(* CODESYS project projeto_final.project

Project tree, tasks and I/O mapping:
  Device : CODESYS Control Win V3, 3S - Smart Software Solutions GmbH, version 3.5.3.50
    application Application
      libraries: Standard, 3.5.2.0 (System)
      task MainTask (cyclic, interval t#20ms, priority 1) calls liga_desliga, projeto_final
      task simula_vagao (cyclic, interval t#10ms, priority 1) calls simula_vagao_descarrega
      task simula_ventilacao (freewheeling, priority 1) calls simula_SA_01_02_ventilacao
      task simula_SA_carregamento (cyclic, interval t#10ms, priority 1) calls simula_SA_01_carregando
      task simula_descarregamento (cyclic, interval t#20ms, priority 1) calls simula_descarga
      program projeto_final [FBD]
      program liga_desliga [LD]
      function block TR_01_transportador_entrada [SFC]: Receber_graos_active, Transfere_graos_active, Passo_inicial_active, Ativa_transferencia_active
      function block vagao_graneleiro [SFC]: Step0_active, Chave_ligada_active, Step1_active, Step2_active, Inicio_active
      function block MG_01_desviador_mangueira [LD]
      function block SA_01_silo_armazenamento [SFC]: Passo_inicial_active, Carrega_silo_active, Descarrega_silo_active, Passo_auxiliar_active, Transfere_moega_active, Liga_alimentador_active
      function block SA_01_02_nivel_silo [FBD]
      program simula_vagao_descarrega [ST]
      program simula_SA_01_02_ventilacao [LD]
      program simula_SA_01_carregando [ST]
      function block SA_02_silo_armazenamento [SFC]: Passo_inicial_active, Passo_auxiliar_active, Carrega_silo_active, Descarrega_silo_active
      program simula_descarga [ST]
  global variables GVL
*)

// GVL
VAR_GLOBAL
	// liga e desliga
	liga        : BOOL;
	liga_local  : BOOL;
	liga_remoto : BOOL;
	seletor_modo: BOOL; // 1 = local e 0 = remoto
	
	// vagao granaleiro
	vagao_chave              : BOOL; // indica que o vagao esta posicionado
	vagao_descarrega         : BOOL; // recebe comando do sistema de supervisao para descarregar
	vagao_capacidade         : INT;  // kg
	vagao_nivel              : INT;
	vagao_taxa_descarrega    : INT;  // kg/s
	vagao_graos_transferidos : INT;
	
	// transportador de entrada TR_01
	TR_01_ligado             : BOOL;
	TR_01_taxa_transferencia : INT;  // 100 kg/s
	TR_01_sensor             : BOOL; // sensor que indica se existe material no transportador
	TR_01_alarme             : BOOL; // se estiver ligado e vazio por mais de 5s
	//TR_01_nivel              : INT;  // kg de graos
	TR_01_carrega			 : BOOL; // indica carregamento
	TR_01_descarrega		 : BOOL; // indica descarregamento
	
	TR_01_SA_graos : INT; // graos que serao transferidos entre o transportador de entrada e dos silos 
	
	// desviador de mangueira
	MG_01_ligado : BOOL; // 
	MG_01_chave  : BOOL; // 0 - primeiro silo 1 - segundo silo
	
	// Silo 1
	SA_01_ligado      : BOOL;
	SA_01_capacidade  : INT;  // 2500
	SA_01_nivel       : INT;  // sensor responsavel por medir o peso do silo
	SA_01_chave_baixo : BOOL; // setada quando o nivel < 100 kg
	SA_01_chave_alto  : BOOL; // setada quando o nivel > 2400 kg
	SA_01_ventilacao  : BOOL; // sistema de ventilacao é ligado quando há carga e descarga
	SA_01_carrega     : BOOL; // silo sendo carregado
	SA_01_descarrega  : BOOL; // silo sendo descarregado
	
	// Silo 2
	SA_02_ligado      : BOOL;
	SA_02_capacidade  : INT;  // 2500
	SA_02_nivel       : INT;  // sensor responsavel por medir o peso do silo
	SA_02_chave_baixo : BOOL; // setada quando o nivel < 100 kg
	SA_02_chave_alto  : BOOL; // setada quando o nivel > 2400 kg
	SA_02_ventilacao  : BOOL; // sistema de ventilacao é ligado quando há carga e descarga
	SA_02_carrega     : BOOL; // silo sendo carregado
	SA_02_descarrega  : BOOL; // silo sendo descarregado
	
	// Alimentadores de moega
	AL_01_ligado      : BOOL; 
	AL_01_taxa_transf : BOOL; // 50 kg/s
	AL_01_sensor      : BOOL; // setado quando há graos no alimentador
	AL_01_alarme      : BOOL; // setado quando ligado e vazio por mais de 5s
	AL_01_nivel       : INT; // graos
	
	AL_02_ligado      : BOOL; 
	AL_02_taxa_transf : BOOL; // 50 kg/s
	AL_02_sensor      : BOOL; // setado quando há graos no alimentador
	AL_02_alarme      : BOOL; // setado quando ligado e vazio por mais de 5s
	AL_02_nivel       : INT; // graos
	
	// Moega de pesagem
	MO_01_ligado : BOOL; // moega ligada
	MO_01_peso   : INT; // contabiliza o peso de graos que esta sendo transferido do silo para o transportador de saida
	MO_01_alarme : BOOL; // ativado quando o transportador de saida está desligado e peso da moega != 0
	
	// Alimentador de saida
	//AL_02_ligado : BOOL; //descarrega graos
	
END_VAR

// Device/Application/liga_desliga
PROGRAM liga_desliga
VAR
END_VAR

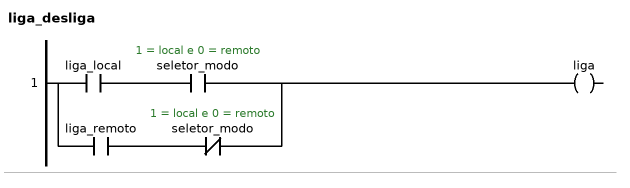
// NETWORK 1
//   seletor_modo: 1 = local e 0 = remoto
liga := liga_local AND seletor_modo OR liga_remoto AND NOT seletor_modo;

END_PROGRAM

// Device/Application/projeto_final
PROGRAM projeto_final
VAR
	vagao_graneleiro_0: vagao_graneleiro;
	TR_01_transportador_entrada_0: TR_01_transportador_entrada;
	MG_01_desviador_mangueira_0: MG_01_desviador_mangueira;
	SA_01_02_nivel_silo_0: SA_01_02_nivel_silo;
	SA_01_silo_armazenamento_0: SA_01_silo_armazenamento;
	SA_02_silo_armazenamento_0: SA_02_silo_armazenamento;
END_VAR

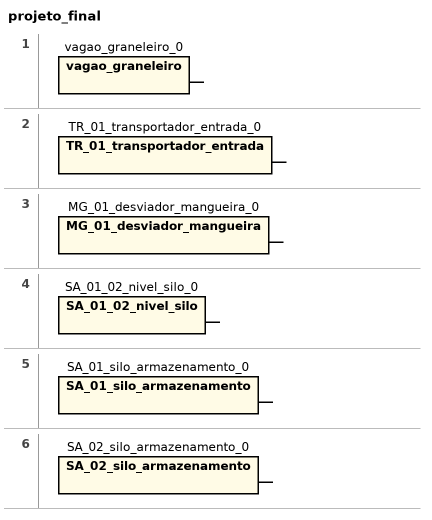
// NETWORK 1
vagao_graneleiro_0(); // vagao_graneleiro

// NETWORK 2
TR_01_transportador_entrada_0(); // TR_01_transportador_entrada

// NETWORK 3
MG_01_desviador_mangueira_0(); // MG_01_desviador_mangueira

// NETWORK 4
SA_01_02_nivel_silo_0(); // SA_01_02_nivel_silo

// NETWORK 5
SA_01_silo_armazenamento_0(); // SA_01_silo_armazenamento

// NETWORK 6
SA_02_silo_armazenamento_0(); // SA_02_silo_armazenamento

END_PROGRAM

// Device/Application/vagao_graneleiro
FUNCTION_BLOCK vagao_graneleiro
VAR_INPUT
END_VAR
VAR_OUTPUT
END_VAR
VAR
END_VAR

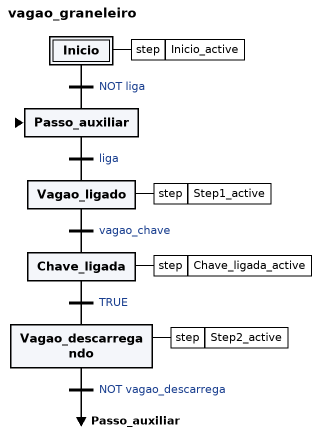
INITIAL_STEP Inicio:
    Inicio_active(N);  // step action
END_STEP
TRANSITION FROM Inicio TO Passo_auxiliar
    := NOT liga;
END_TRANSITION
STEP Passo_auxiliar:
END_STEP
TRANSITION FROM Passo_auxiliar TO Vagao_ligado
    := liga;
END_TRANSITION
STEP Vagao_ligado:
    Step1_active(N);  // step action
END_STEP
TRANSITION FROM Vagao_ligado TO Chave_ligada
    := vagao_chave;
END_TRANSITION
STEP Chave_ligada:
    Chave_ligada_active(N);  // step action
END_STEP
TRANSITION FROM Chave_ligada TO Vagao_descarregando
    := TRUE;
END_TRANSITION
STEP Vagao_descarregando:
    Step2_active(N);  // step action
END_STEP
TRANSITION FROM Vagao_descarregando TO Passo_auxiliar
    := NOT vagao_descarrega;
END_TRANSITION

ACTION Step0_active:
vagao_nivel := vagao_capacidade;
END_ACTION

ACTION Chave_ligada_active:
vagao_descarrega := 1;
END_ACTION

ACTION Step1_active:
vagao_nivel := vagao_capacidade;
END_ACTION

ACTION Step2_active:
vagao_chave := 0;
END_ACTION

ACTION Inicio_active:
vagao_capacidade := 1000;
vagao_taxa_descarrega := 100;
vagao_graos_transferidos := 0;
END_ACTION

END_FUNCTION_BLOCK

// Device/Application/TR_01_transportador_entrada
FUNCTION_BLOCK TR_01_transportador_entrada
VAR_INPUT
END_VAR
VAR_OUTPUT
END_VAR
VAR
END_VAR

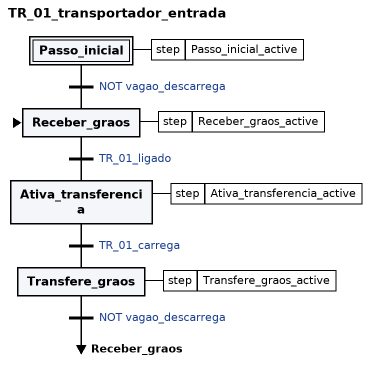
INITIAL_STEP Passo_inicial:
    Passo_inicial_active(N);  // step action
END_STEP
TRANSITION FROM Passo_inicial TO Receber_graos
    := NOT vagao_descarrega;
END_TRANSITION
STEP Receber_graos:
    Receber_graos_active(N);  // step action
END_STEP
TRANSITION FROM Receber_graos TO Ativa_transferencia
    := TR_01_ligado;
END_TRANSITION
STEP Ativa_transferencia:
    Ativa_transferencia_active(N);  // step action
END_STEP
TRANSITION FROM Ativa_transferencia TO Transfere_graos
    := TR_01_carrega;
END_TRANSITION
STEP Transfere_graos:
    Transfere_graos_active(N);  // step action
END_STEP
TRANSITION FROM Transfere_graos TO Receber_graos
    := NOT vagao_descarrega;
END_TRANSITION

ACTION Receber_graos_active:
TR_01_ligado := 1;
//TR_01_nivel := vagao_graos_transferidos;
END_ACTION

ACTION Transfere_graos_active:

END_ACTION

ACTION Passo_inicial_active:
TR_01_taxa_transferencia := 100; // 100 kg/s
END_ACTION

ACTION Ativa_transferencia_active:

END_ACTION

END_FUNCTION_BLOCK

// Device/Application/MG_01_desviador_mangueira
FUNCTION_BLOCK MG_01_desviador_mangueira
VAR_INPUT
END_VAR
VAR_OUTPUT
END_VAR
VAR
END_VAR

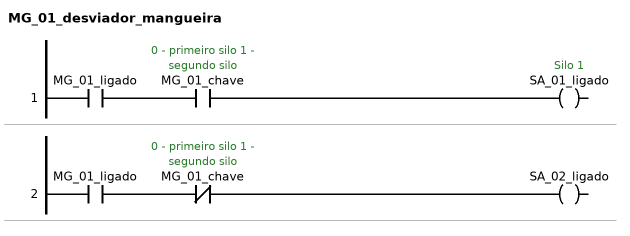
// NETWORK 1
//   MG_01_chave: 0 - primeiro silo 1 - segundo silo
//   SA_01_ligado: Silo 1
SA_01_ligado := MG_01_ligado AND MG_01_chave;

// NETWORK 2
//   MG_01_chave: 0 - primeiro silo 1 - segundo silo
SA_02_ligado := MG_01_ligado AND NOT MG_01_chave;

END_FUNCTION_BLOCK

// Device/Application/SA_01_02_nivel_silo
FUNCTION_BLOCK SA_01_02_nivel_silo
VAR_INPUT
END_VAR
VAR_OUTPUT
END_VAR
VAR
END_VAR

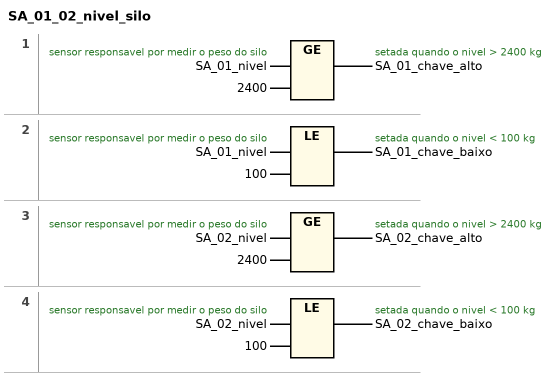
// NETWORK 1
//   SA_01_nivel: sensor responsavel por medir o peso do silo
//   SA_01_chave_alto: setada quando o nivel > 2400 kg
SA_01_chave_alto := SA_01_nivel >= 2400;

// NETWORK 2
//   SA_01_nivel: sensor responsavel por medir o peso do silo
//   SA_01_chave_baixo: setada quando o nivel < 100 kg
SA_01_chave_baixo := SA_01_nivel <= 100;

// NETWORK 3
//   SA_02_nivel: sensor responsavel por medir o peso do silo
//   SA_02_chave_alto: setada quando o nivel > 2400 kg
SA_02_chave_alto := SA_02_nivel >= 2400;

// NETWORK 4
//   SA_02_nivel: sensor responsavel por medir o peso do silo
//   SA_02_chave_baixo: setada quando o nivel < 100 kg
SA_02_chave_baixo := SA_02_nivel <= 100;

END_FUNCTION_BLOCK

// Device/Application/SA_01_silo_armazenamento
FUNCTION_BLOCK SA_01_silo_armazenamento
VAR_INPUT
END_VAR
VAR_OUTPUT
END_VAR
VAR
END_VAR

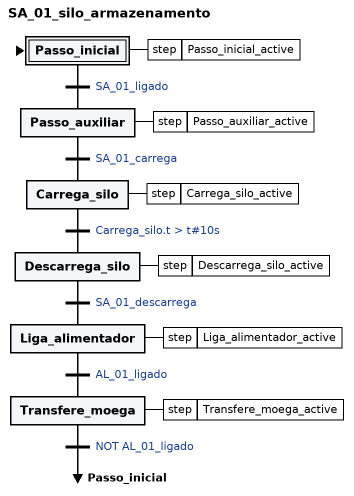
INITIAL_STEP Passo_inicial:
    Passo_inicial_active(N);  // step action
END_STEP
TRANSITION FROM Passo_inicial TO Passo_auxiliar
    := SA_01_ligado;
END_TRANSITION
STEP Passo_auxiliar:
    Passo_auxiliar_active(N);  // step action
END_STEP
TRANSITION FROM Passo_auxiliar TO Carrega_silo
    := SA_01_carrega;
END_TRANSITION
STEP Carrega_silo:
    Carrega_silo_active(N);  // step action
END_STEP
TRANSITION FROM Carrega_silo TO Descarrega_silo
    := Carrega_silo.t > t#10s;
END_TRANSITION
STEP Descarrega_silo:
    Descarrega_silo_active(N);  // step action
END_STEP
TRANSITION FROM Descarrega_silo TO Liga_alimentador
    := SA_01_descarrega;
END_TRANSITION
STEP Liga_alimentador:
    Liga_alimentador_active(N);  // step action
END_STEP
TRANSITION FROM Liga_alimentador TO Transfere_moega
    := AL_01_ligado;
END_TRANSITION
STEP Transfere_moega:
    Transfere_moega_active(N);  // step action
END_STEP
TRANSITION FROM Transfere_moega TO Passo_inicial
    := NOT AL_01_ligado;
END_TRANSITION

ACTION Passo_inicial_active:
SA_01_capacidade := 2500;
END_ACTION

ACTION Carrega_silo_active:
SA_01_nivel := vagao_graos_transferidos;
END_ACTION

ACTION Descarrega_silo_active:
vagao_graos_transferidos := 0;
SA_01_descarrega := 1;
SA_01_ligado := 0;
SA_01_carrega := 0;
MG_01_ligado := 0;
MG_01_chave  := 0;
END_ACTION

ACTION Passo_auxiliar_active:
SA_01_carrega := 1;
END_ACTION

ACTION Transfere_moega_active:

END_ACTION

ACTION Liga_alimentador_active:
AL_01_ligado := 1;
END_ACTION

END_FUNCTION_BLOCK

// Device/Application/SA_02_silo_armazenamento
FUNCTION_BLOCK SA_02_silo_armazenamento
VAR_INPUT
END_VAR
VAR_OUTPUT
END_VAR
VAR
END_VAR

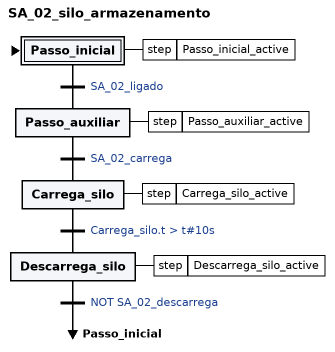
INITIAL_STEP Passo_inicial:
    Passo_inicial_active(N);  // step action
END_STEP
TRANSITION FROM Passo_inicial TO Passo_auxiliar
    := SA_02_ligado;
END_TRANSITION
STEP Passo_auxiliar:
    Passo_auxiliar_active(N);  // step action
END_STEP
TRANSITION FROM Passo_auxiliar TO Carrega_silo
    := SA_02_carrega;
END_TRANSITION
STEP Carrega_silo:
    Carrega_silo_active(N);  // step action
END_STEP
TRANSITION FROM Carrega_silo TO Descarrega_silo
    := Carrega_silo.t > t#10s;
END_TRANSITION
STEP Descarrega_silo:
    Descarrega_silo_active(N);  // step action
END_STEP
TRANSITION FROM Descarrega_silo TO Passo_inicial
    := NOT SA_02_descarrega;
END_TRANSITION

ACTION Passo_inicial_active:
SA_02_capacidade := 2500;
END_ACTION

ACTION Passo_auxiliar_active:
SA_02_carrega := 1;
END_ACTION

ACTION Carrega_silo_active:
SA_02_nivel := vagao_graos_transferidos;
END_ACTION

ACTION Descarrega_silo_active:
vagao_graos_transferidos := 0;
SA_02_descarrega := 1;
SA_02_ligado := 0;
SA_02_carrega := 0;
MG_01_ligado := 0;
MG_01_chave  := 0;
END_ACTION

END_FUNCTION_BLOCK

// Device/Application/simula_vagao_descarrega
PROGRAM simula_vagao_descarrega
VAR
END_VAR

IF(vagao_descarrega) THEN
	vagao_nivel := vagao_nivel - 1;
	vagao_graos_transferidos := vagao_graos_transferidos + 1;
	IF(vagao_nivel = 0) THEN
		vagao_descarrega := 0;
	END_IF
END_IF

END_PROGRAM

// Device/Application/simula_SA_01_02_ventilacao
PROGRAM simula_SA_01_02_ventilacao
VAR
END_VAR

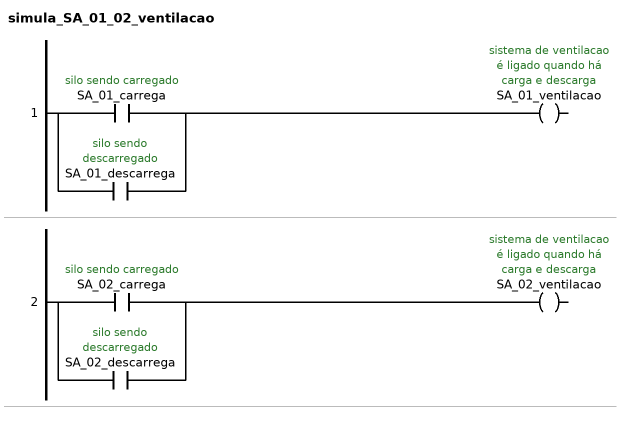
// NETWORK 1
//   SA_01_carrega: silo sendo carregado
//   SA_01_descarrega: silo sendo descarregado
//   SA_01_ventilacao: sistema de ventilacao é ligado quando há carga e descarga
SA_01_ventilacao := SA_01_carrega OR SA_01_descarrega;

// NETWORK 2
//   SA_02_carrega: silo sendo carregado
//   SA_02_descarrega: silo sendo descarregado
//   SA_02_ventilacao: sistema de ventilacao é ligado quando há carga e descarga
SA_02_ventilacao := SA_02_carrega OR SA_02_descarrega;

END_PROGRAM

// Device/Application/simula_SA_01_carregando
PROGRAM simula_SA_01_carregando
VAR
END_VAR

//IF (SA_01_carrega) THEN
//	vagao_graos_transferidos := vagao_graos_transferidos - 1;
	//SA_01_nivel := SA_01_nivel + 1;
	//IF(SA_01_nivel >= 1000) THEN
		//SA_01_carrega := 0;
	//	SA_01_descarrega := 1;
	//END_IF
	//IF(vagao_graos_transferidos <= 0) THEN
	//	SA_01_carrega := 0;
	//END_IF
//END_IF

END_PROGRAM

// Device/Application/simula_descarga
PROGRAM simula_descarga
VAR
END_VAR

IF(AL_01_ligado) THEN	
	SA_01_nivel := SA_01_nivel - 1;
	AL_01_nivel := AL_01_nivel + 1;
	MO_01_peso := MO_01_peso + 1;
	IF(SA_01_nivel <= 0) THEN
		AL_01_ligado := 0;
	END_IF
END_IF

END_PROGRAM
